// TIA Portal V20 export
VAR_GLOBAL   // PLC tag table "Unit1Em5_Servo"
   "BA030AZSBK07.00" AT %I1024.0 : Bool;   // CATHODE MAIN P&P1 Z-AXIS LIMIT SENSOR(-)
   "BA030AZSBK07.01" AT %I1024.1 : Bool;   // CATHODE MAIN P&P1 Z-AXIS LIMIT SENSOR(+)
   "BA030AZSBK07.02" AT %I1024.2 : Bool;   // CATHODE MAIN P&P1 Y-AXIS LIMIT SENSOR(-)
   "BA030AZSBK07.03" AT %I1024.3 : Bool;   // CATHODE MAIN P&P1 Y-AXIS LIMIT SENSOR(+)
   "BA030AZSBK07.10" AT %I1025.0 : Bool;   // CATHODE MAIN P&P1 Z-AXIS HOME SENSOR
   "BA030AZSBK07.12" AT %I1025.2 : Bool;   // CATHODE MAIN P&P1 Y-AXIS HOME SENSOR
   "BA030AZSBK08.00" AT %I1028.0 : Bool;   // CATHODE MAIN P&P2 Z-AXIS LIMIT SENSOR(-)
   "BA030AZSBK08.01" AT %I1028.1 : Bool;   // CATHODE MAIN P&P2 Z-AXIS HOME SENSOR
   "BA030AZSBK08.02" AT %I1028.2 : Bool;   // CATHODE MAIN P&P2 Z-AXIS LIMIT SENSOR(+)
   "BA030AZSBK13.01" AT %I1048.1 : Bool;   // CATHODE ALIGN TABLE X-AXIS LIMIT SENSOR(+)
   "BA030AZSBK13.00" AT %I1048.0 : Bool;   // CATHODE ALIGN TABLE X-AXIS LIMIT SENSOR(-)
   "BA030AZSBK13.02" AT %I1048.2 : Bool;   // CATHODE ALIGN TABLE Y1-AXIS LIMIT SENSOR(-)
   "BA030AZSBK13.03" AT %I1048.3 : Bool;   // CATHODE ALIGN TABLE Y1-AXIS LIMIT SENSOR(+)
   "BA030AZSBK13.04" AT %I1048.4 : Bool;   // CATHODE ALIGN TABLE Y2-AXIS LIMIT SENSOR(-)
   "BA030AZSBK13.05" AT %I1048.5 : Bool;   // CATHODE ALIGN TABLE Y2-AXIS LIMIT SENSOR(+)
   "BA030AZSBK13.12" AT %I1049.2 : Bool;   // CATHODE ALIGN TABLE Y1-AXIS HOME SENSOR
   "BA030AZSBK13.14" AT %I1049.4 : Bool;   // CATHODE ALIGN TABLE Y2-AXIS HOME SENSOR
   "BA030AZSBK13.10" AT %I1049.0 : Bool;   // CATHODE ALIGN TABLE X-AXIS HOME SENSOR
   "BA030AZSBK04.02" AT %I1012.2 : Bool;   // CATHODE MAIN P&P1 X-AXIS LIMITS SENSOR(-)
   "BA030AZSBK04.03" AT %I1012.3 : Bool;   // CATHODE MAIN P&P1 X-AXIS LIMITS SENSOR(+)
   "BA030AZSBK04.12" AT %I1013.2 : Bool;   // CATHODE MAIN P&P1 X-AXIS LIMITS SENSOR HOME
   "BA030AZSBK04.06" AT %I1012.6 : Bool;   // CATHODE MAIN P&P2 X-AXIS LIMITS SENSOR(-)
   "BA030AZSBK04.07" AT %I1012.7 : Bool;   // CATHODE MAIN P&P2 X-AXIS LIMITS SENSOR(+)
   "BA030AZSBK04.16" AT %I1013.6 : Bool;   // CATHODE MAIN P&P2 X-AXIS LIMITS SENSOR HOME
END_VAR
